// TIA Portal V20 export
TYPE "LBP_typeMcp483PnOutput"
TITLE = MCP 483 PN image / Image du MCP 483 PN
// Output image of MCP 483 PN / Image de sortie du MCP 483 PN
   STRUCT
      standard { S7_SetPoint := 'True'} : "LBP_typeMcp483StandardOutput";   // Output image of MCP 483 / Image de sortie du MCP 483
   END_STRUCT;
END_TYPE
